{attribute 'qualified_only'}
{attribute 'strict'}
{attribute 'to_string'}
TYPE sensorID_t :
(
	EXPANTION_SENSOR_X0_0 := 0, 
	EXPANTION_SENSOR_X0_1,
	
	EXPANTION_SENSOR_X1_0, 
	EXPANTION_SENSOR_X1_1,
	
	EXPANTION_SENSOR_X2_0, 
	EXPANTION_SENSOR_X2_1,
	
	EXPANTION_SENSOR_X3_0, 
	EXPANTION_SENSOR_X3_1,
	
	EXPANTION_SENSOR_X4_0, 
	EXPANTION_SENSOR_X4_1,
	
	EXPANTION_SENSOR_X5_0, 
	EXPANTION_SENSOR_X5_1,
	
	EXPANTION_SENSOR_X6_0, 
	EXPANTION_SENSOR_X6_1,
	
	EXPANTION_SENSOR_X7_0, 
	EXPANTION_SENSOR_X7_1,
	
	SENSOR_X6_0,
	SENSOR_X6_1
);
END_TYPE

(* stored: Version 1.1.0.1
   EnumerationTextList sensorID_t: Id {f89e3e14-12ca-4816-bc72-26eced312805} *)
